// TIA Portal V19 export
TYPE "A0301_Mach_Sens_Par"
   STRUCT
      Tol_Work { S7_SetPoint := 'True'} : Real;   // Valore di tolleranza di lavoro
      WorkTime_SensDisable { S7_SetPoint := 'True'} : Time;
   END_STRUCT;
END_TYPE
